PROGRAM MAIN
VAR
END_VAR

F_ConsumeTime(100);

END_PROGRAM

(* stored: Version 1.1.0.1, ProductVersion 3.1.4026.18
   POU MAIN: Id {c533c4a0-a466-4576-8630-c01f6db1c0bc}, SpecialFunc None *)
